# EPICS substitutions: acqirisApp/Db/userHost.substitutions
# Example substitutions file

file "db/dbExample1.db" {
    { user = "yhuHost" }
}

file db/dbExample2.db {
    pattern { user, no, scan }
        { "yhuHost", 1, "1 second" }
        { "yhuHost", 2, "2 second" }
        { "yhuHost", 3, "5 second" }
}
